FUNCTION_BLOCK FB_CurrentTime
VAR_INPUT
	fbTime   : FB_LocalSystemTime := ( bEnable := TRUE, dwCycle := 1 );
END_VAR
VAR_OUTPUT
END_VAR
VAR
	currH : WORD;
	currM : WORD;
	currD : WORD;
	CurrDate: WORD;
END_VAR

fbTime();
currH := fbTime.systemTime.wHour;
currM := fbTime.systemTime.wMinute;
currD := fbTime.systemTime.wDayOfWeek;
CurrDate := fbTime.systemTime.wDay;

END_FUNCTION_BLOCK

(* stored: Version 1.1.0.1, ProductVersion 3.1.4024.14
   POU FB_CurrentTime: Id {046edf5d-f138-4d66-a903-c153b324f3d9}, SpecialFunc None *)
